// TIA Portal V17 export
// export: Created 2025-08-05T09:36:00.1023537Z, ExportSetting WithDefaults, DisplayName Totally Integrated Automation Portal, DisplayVersion V17, DisplayName TIA Portal Openness, DisplayVersion V17, DisplayName TIA Portal Version Control Interface, DisplayVersion V17, DisplayName SINAMICS Startdrive Advanced, DisplayVersion V17, DisplayName SINAMICS Startdrive G130, G150, S120, S150, SINAMICS MV, S210, DisplayVersion V17, DisplayName SINAMICS Startdrive G110M, G120, G120C, G120D, G120P, G115D, DisplayVersion V17, DisplayName STEP 7 Professional, DisplayVersion V17, DisplayName STEP 7 Safety, DisplayVersion V17, DisplayName WinCC Advanced, DisplayVersion V17
TYPE "typeHmiManualGroup"
TITLE = HMI setup groups / HMI Einricht Gruppen
// HMI Setup groups [V 01.00 | Kernel_V2] / HMI Einricht Gruppen [V 01.00 | Kernel_V2]
// stored: IsFailsafeCompliant false
   STRUCT
      selectedGroup : Array[1..30] of Bool;   // Gruppe Handbedienbild / Group manual operating screen
      manualButtonRight : Bool;   // rechte Taste gedrückt / Right key pressed
      manualButtonLeft : Bool;   // linke Taste gedrückt / Left key pressed
   END_STRUCT;
END_TYPE
